PROGRAM POU
VAR
END_VAR

END_PROGRAM

(* stored: Version 1.1.0.1, ProductVersion 3.1.4024.12
   POU POU: Id {79a7a6b2-14ff-42b1-9d57-fc152064c40b}, SpecialFunc None *)
